// Mitsubishi GX Works2 project: IELET2103_Øving3   PLC: FX2N/FX2NC
// IELET2103_Øving3

// global labels: Global1
VAR_GLOBAL
  seq : INT;
  Start AT M100 : BOOL;
  Stopp AT M101 : BOOL;
  Dreieretning AT M102 : BOOL;
  Modulplass0 : INT;
  Brukstimer : WORD;
  D15output AT D60 : ARRAY [0..1] OF DINT;
  vektor AT D0 : ARRAY [0..19] OF INT;
  D10annenhver : INT;
  Varsellampe AT Y000 : BOOL;
  Start_Stopp AT Y001 : BOOL;
  Medurs AT Y002 : BOOL;
  Moturs AT Y003 : BOOL;
END_VAR

// task Task_01 (event TRUE, interval 0, priority 31): Oppgave3

PROGRAM Oppgave1a)
VAR
  TON_1 : TON;
  tid : WORD;
END_VAR
(* structured ladder/FBD written out as ST: instructions are called as NAME(EN, inputs, outputs); _pN, _eN, _tN stand for wires *)
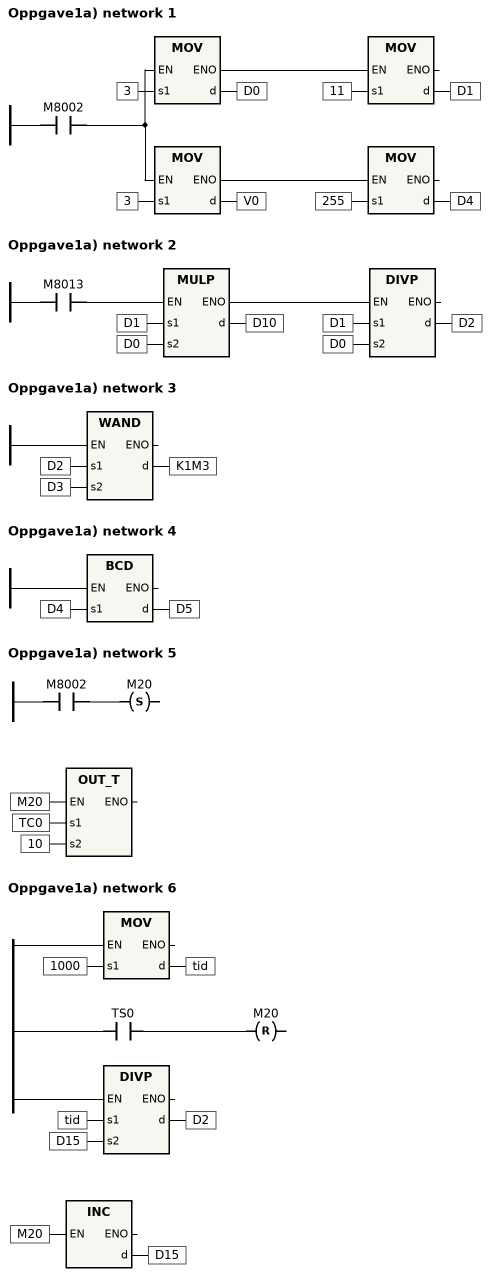
(* network 1 *)
_e1 := MOV(M8002, 3, D0);
MOV(_e1, 11, D1);
_e2 := MOV(M8002, 3, V0);
MOV(_e2, 255, D4);
(* network 2 *)
_e1 := MULP(M8013, D1, D0, D10);
DIVP(_e1, D1, D0, D2);
(* network 3 *)
WAND(TRUE, D2, D3, K1M3);
(* network 4 *)
BCD(TRUE, D4, D5);
(* network 5 *)
SET(M8002, M20);
OUT_T(M20, TC0, 10);
(* network 6 *)
RST(TS0, M20);
INC(M20, D15);
MOV(TRUE, 1000, tid);
DIVP(TRUE, tid, D15, D2);
END_PROGRAM

PROGRAM Oppgave1b)
VAR
  D15tmp : DINT;
END_VAR
(* structured ladder/FBD written out as ST: instructions are called as NAME(EN, inputs, outputs); _pN, _eN, _tN stand for wires *)
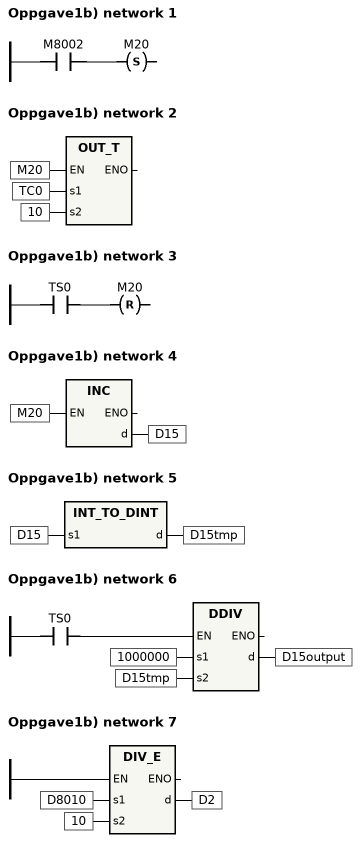
(* network 1 *)
SET(M8002, M20);
(* network 2 *)
OUT_T(M20, TC0, 10);
(* network 3 *)
RST(TS0, M20);
(* network 4 *)
INC(M20, D15);
(* network 5 *)
D15tmp := INT_TO_DINT(D15);
(* network 6 *)
DDIV(TS0, 1000000, D15tmp, D15output);
(* network 7 *)
DIV_E(TRUE, D8010, 10, D2);
END_PROGRAM

PROGRAM Oppgave1c)
(* structured ladder/FBD written out as ST: instructions are called as NAME(EN, inputs, outputs); _pN, _eN, _tN stand for wires *)
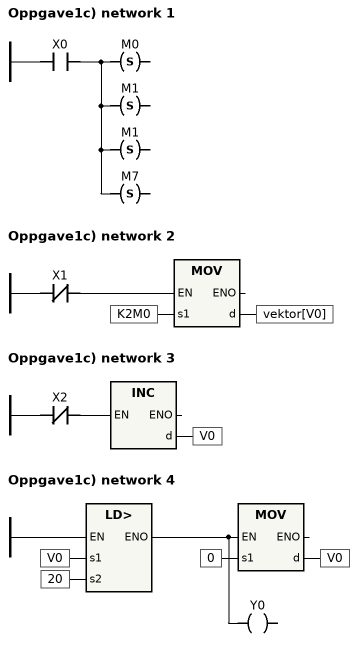
(* network 1 *)
SET(X0, M0);
SET(X0, M1);
SET(X0, M1);
SET(X0, M7);
(* network 2 *)
MOV(NOT X1, K2M0, vektor[V0]);
(* network 3 *)
INC(NOT X2, V0);
(* network 4 *)
_e1 := LD>(TRUE, V0, 20);
Y0 := _e1;
MOV(_e1, 0, V0);
END_PROGRAM

PROGRAM Oppgave1d)
(* structured ladder/FBD written out as ST: instructions are called as NAME(EN, inputs, outputs); _pN, _eN, _tN stand for wires *)
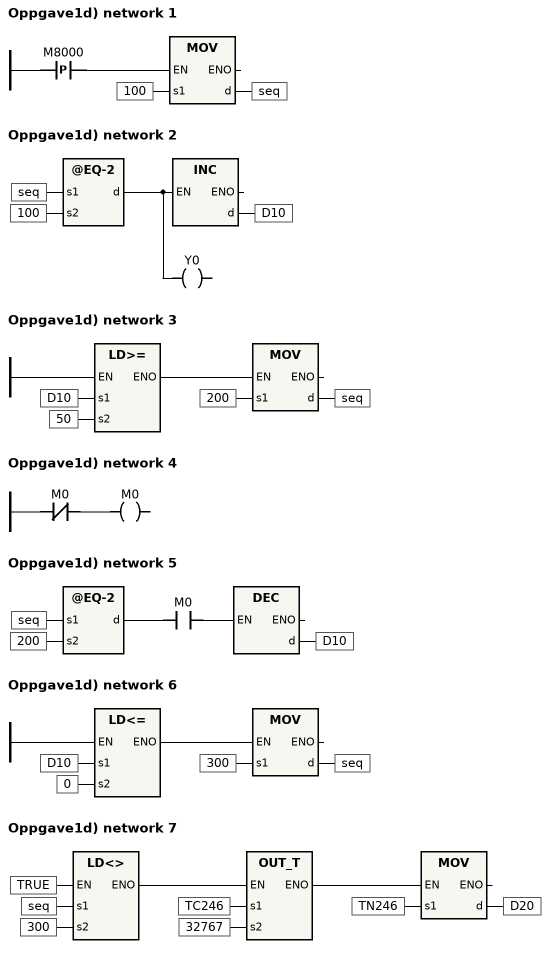
(* network 1 *)
MOV(LDP(TRUE, M8000), 100, seq);
(* network 2 *)
_p1 := @EQ-2(seq, 100);
INC(_p1, D10);
Y0 := _p1;
(* network 3 *)
_e1 := LD>=(TRUE, D10, 50);
MOV(_e1, 200, seq);
(* network 4 *)
M0 := NOT M0;
(* network 5 *)
DEC(@EQ-2(seq, 200) AND M0, D10);
(* network 6 *)
_e1 := LD<=(TRUE, D10, 0);
MOV(_e1, 300, seq);
(* network 7 *)
_e1 := LD<>(TRUE, seq, 300);
_e2 := OUT_T(_e1, TC246, 32767);
MOV(_e2, TN246, D20);
END_PROGRAM

PROGRAM Oppgave2
VAR
  D0tmp : INT;
END_VAR
(* structured ladder/FBD written out as ST: instructions are called as NAME(EN, inputs, outputs); _pN, _eN, _tN stand for wires *)
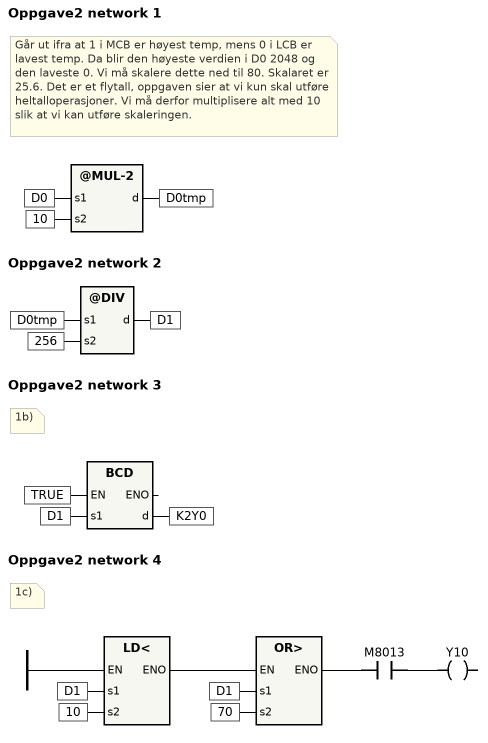
(* network 1 *)
(* Går ut ifra at 1 i MCB er høyest temp, mens 0 i LCB er lavest temp. Da blir den høyeste verdien i D0 2048 og den laveste 0. Vi må skalere dette ned til 80. Skalaret er 25.6. Det er et flytall, oppgaven sier at vi kun skal utføre heltalloperasjoner. Vi må derfor multiplisere alt med 10 slik at vi kan utføre skaleringen. *)
D0tmp := @MUL-2(D0, 10);
(* network 2 *)
D1 := @DIV(D0tmp, 256);
(* network 3 *)
(* 1b) *)
BCD(TRUE, D1, K2Y0);
(* network 4 *)
(* 1c) *)
_e1 := LD<(TRUE, D1, 10);
_e2 := OR>(_e1, D1, 70);
Y10 := _e2 AND M8013;
END_PROGRAM

PROGRAM Oppgave3
VAR
  D100tmp : INT;
  D100DW : DINT;
END_VAR
(* structured ladder/FBD written out as ST: instructions are called as NAME(EN, inputs, outputs); _pN, _eN, _tN stand for wires *)
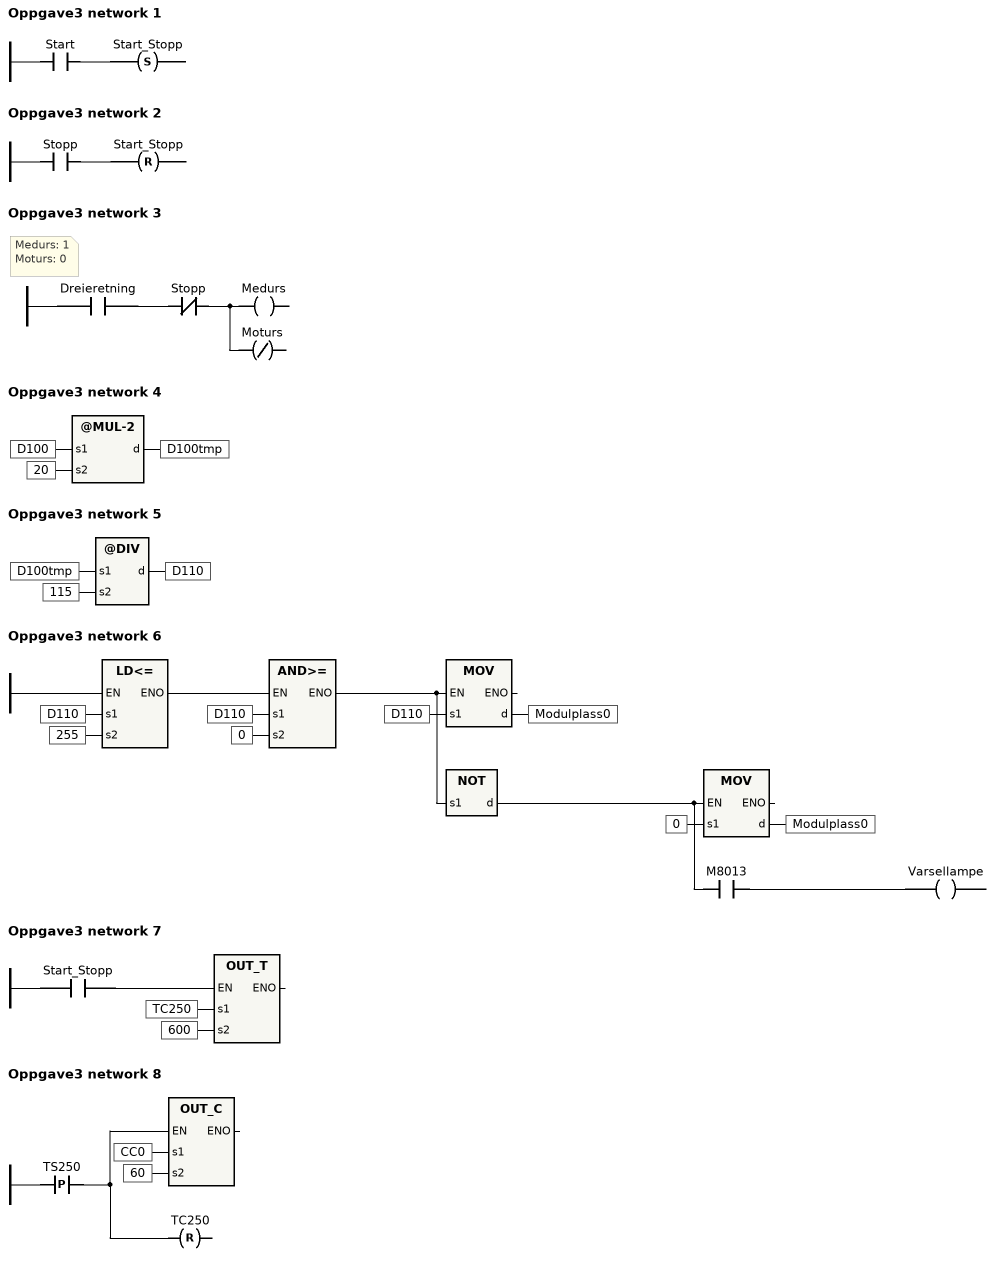
(* network 1 *)
SET(Start, Start_Stopp);
(* network 2 *)
RST(Stopp, Start_Stopp);
(* network 3 *)
(* Medurs: 1 / Moturs: 0 *)
_p1 := Dreieretning AND NOT Stopp;
Medurs := _p1;
Moturs := NOT _p1;
(* network 4 *)
D100tmp := @MUL-2(D100, 20);
(* network 5 *)
D110 := @DIV(D100tmp, 115);
(* network 6 *)
_e1 := LD<=(TRUE, D110, 255);
_e2 := AND>=(_e1, D110, 0);
MOV(_e2, D110, Modulplass0);
_p3 := NOT(_e2);
Varsellampe := _p3 AND M8013;
MOV(_p3, 0, Modulplass0);
(* network 7 *)
OUT_T(Start_Stopp, TC250, 600);
(* network 8 *)
_p1 := LDP(TRUE, TS250);
OUT_C(_p1, CC0, 60);
RST(_p1, TC250);
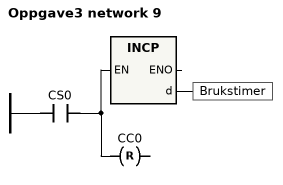
(* network 9 *)
INCP(CS0, Brukstimer);
RST(CS0, CC0);
END_PROGRAM
